// TIA Portal V17 export
// export: Created 2025-07-01T14:26:18.6925672Z, ExportSetting WithDefaults, DisplayName Totally Integrated Automation Portal, DisplayVersion V17 Update 8, DisplayName TIA Portal Openness, DisplayVersion V17 Update 8, DisplayName TIA Portal Version Control Interface, DisplayVersion V17, DisplayName SINAMICS Startdrive Advanced, DisplayVersion V17 SP2, DisplayName SINAMICS Startdrive G110M, G120, G120C, G120D, G120P, G115D, DisplayVersion V17 SP2, DisplayName SINAMICS Startdrive G130, G150, S120, S150, SINAMICS MV, S210, DisplayVersion V17 SP2, DisplayName STEP 7 Professional, DisplayVersion V17 Update 8, DisplayName SINUMERIK ONE STEP 7 Toolbox, DisplayVersion V17 Update 12, DisplayName SINUMERIK ONE PLC Basic Program Plus, DisplayVersion V17 Update 12, DisplayName SINUMERIK 840D sl STEP 7 Toolbox, DisplayVersion V17 Update 12, DisplayName STEP 7 Safety, DisplayVersion V17 Update 6, DisplayName WinCC Advanced, DisplayVersion V17 Update 8
DATA_BLOCK "DB442_MACHINE_RUN_OUT_ALARM_DECODING"   // DB442
{ S7_Optimized_Access := 'FALSE'; DB_Accessible_From_OPC_UA := 'FALSE' }
AUTHOR : ETXETAR
VERSION : 1.0
// stored: AutoNumber false, DBAccessibleFromOPCUA false, DBAccessibleFromWebserver true, IsOnlyStoredInLoadMemory false, IsWriteProtectedInAS false
   VAR RETAIN
      GLOBAL : Struct
         ANY_RHP_RO_ACTIVE : Bool;   // ANY RETURN HOME POSITION RUN OUT ALARM ACTIVE
         ANY_SEOC_RO_ACTIVE : Bool;   // ANY STOP END OF CYCLE RUN OUT ALARM ACTIVE
         ANY_RO_ACTIVE : Bool;   // ANY RUN OUT ALARM ACTIVE
      END_STRUCT;
      GENERAL : Struct
         RO_ALARMS : Bool;   // GENERAL RUN OUT ALARM
      END_STRUCT;
      UNIT_1 : Struct
         STATION_0 : "RUN_OUT_ALARM";
         STATION_1 : "RUN_OUT_ALARM";
         STATION_2 : "RUN_OUT_ALARM";
         STATION_3 : "RUN_OUT_ALARM";
         STATION_4 : "RUN_OUT_ALARM";
         ALARM_RESET_LOCAL_SEQ_AUX : Struct
            STATION_0 : Bool;
            STATION_1 : Bool;
            STATION_2 : Bool;
            STATION_3 : Bool;
            STATION_4 : Bool;
            PULSES : Array[0..15] of Bool;
         END_STRUCT;
      END_STRUCT;
      UNIT_2 : Struct
         STATION_0 : "RUN_OUT_ALARM";
         STATION_1 : "RUN_OUT_ALARM";
         STATION_2 : "RUN_OUT_ALARM";
         STATION_3 : "RUN_OUT_ALARM";
         STATION_4 : "RUN_OUT_ALARM";
         ALARM_RESET_LOCAL_SEQ_AUX : Struct
            STATION_0 : Bool;
            STATION_1 : Bool;
            STATION_2 : Bool;
            STATION_3 : Bool;
            STATION_4 : Bool;
            PULSES : Array[0..15] of Bool;
         END_STRUCT;
      END_STRUCT;
      UNIT_3 : Struct
         CONTROL_STATION : "RUN_OUT_ALARM";
         ALARM_RESET_LOCAL_SEQ_AUX : Struct
            CONTROL_STATION : Bool;
            PULSES : Array[0..15] of Bool;
         END_STRUCT;
      END_STRUCT;
      ALARM_DECODING : DInt;   // PROGRAMMING ALARM DECODING
      TIMER_ALARMS_DELAY { S7_SetPoint := 'True'} : TON_TIME;
   END_VAR
BEGIN
   TIMER_ALARMS_DELAY.PT := T#3s;
END_DATA_BLOCK
